(* Schneider Machine Expert - Basic project Ladder_Code, file version 2.7.0.0 *)
(* ProjectInformations: Name=New project *)

HARDWARE
  Cpu 0: TM200CE40R
  EthernetConfiguration: NetworkName=M200, IpAllocationMode=FixedAddress, IpAddress=192.168.1.200, SubnetMask=255.255.255.0
  SerialLineConfiguration: Baud=Baud19200, Parity=ParityEven, DataBits=DataBits8, StopBits=StopBits1, PhysicalMedium=PhysicalMediumRs485, TransmissionMode=TransmissionModeModbusRtu, SlaveId=1, Addressing=MasterAddressing
  MastTask: UsePeriodScanMode=false, PeriodScan=100
  FastTask: Period=255
  CpuBehavior: StartingMode=StartAsPreviousState, AutoSaveRamOnEeprom=true, WatchdogPeriod=250

SYMBOLS  (address, symbol, comment, settings)
  %TM0        [Type=TP, Preset=1, Base=OneHundredMilliSeconds]
  %TM1        [Type=TP, Preset=1, Base=OneHundredMilliSeconds]
  %READ_VAR0   [Link(Value(FBComLinkParameterEnums=SerialLine1)), RemoteDeviceId(Value(int=1)), Timeout(Value(int=100)), ObjType(Value(FBComObjTypeParameterEnums=MW)), FirstObj(Value(int=0)), Quantity(Value(int=1)), IndexData(Value(int=100))]
  %WRITE_VAR0   [Link(Value(FBComLinkParameterEnums=SerialLine1)), RemoteDeviceId(Value(int=1)), Timeout(Value(int=100)), ObjType(Value(FBComObjTypeParameterEnums=MW)), FirstObj(Value(int=1)), Quantity(Value(int=1)), IndexData(Value(int=1))]

POU New POU
  (* SectionNumber=1 *)

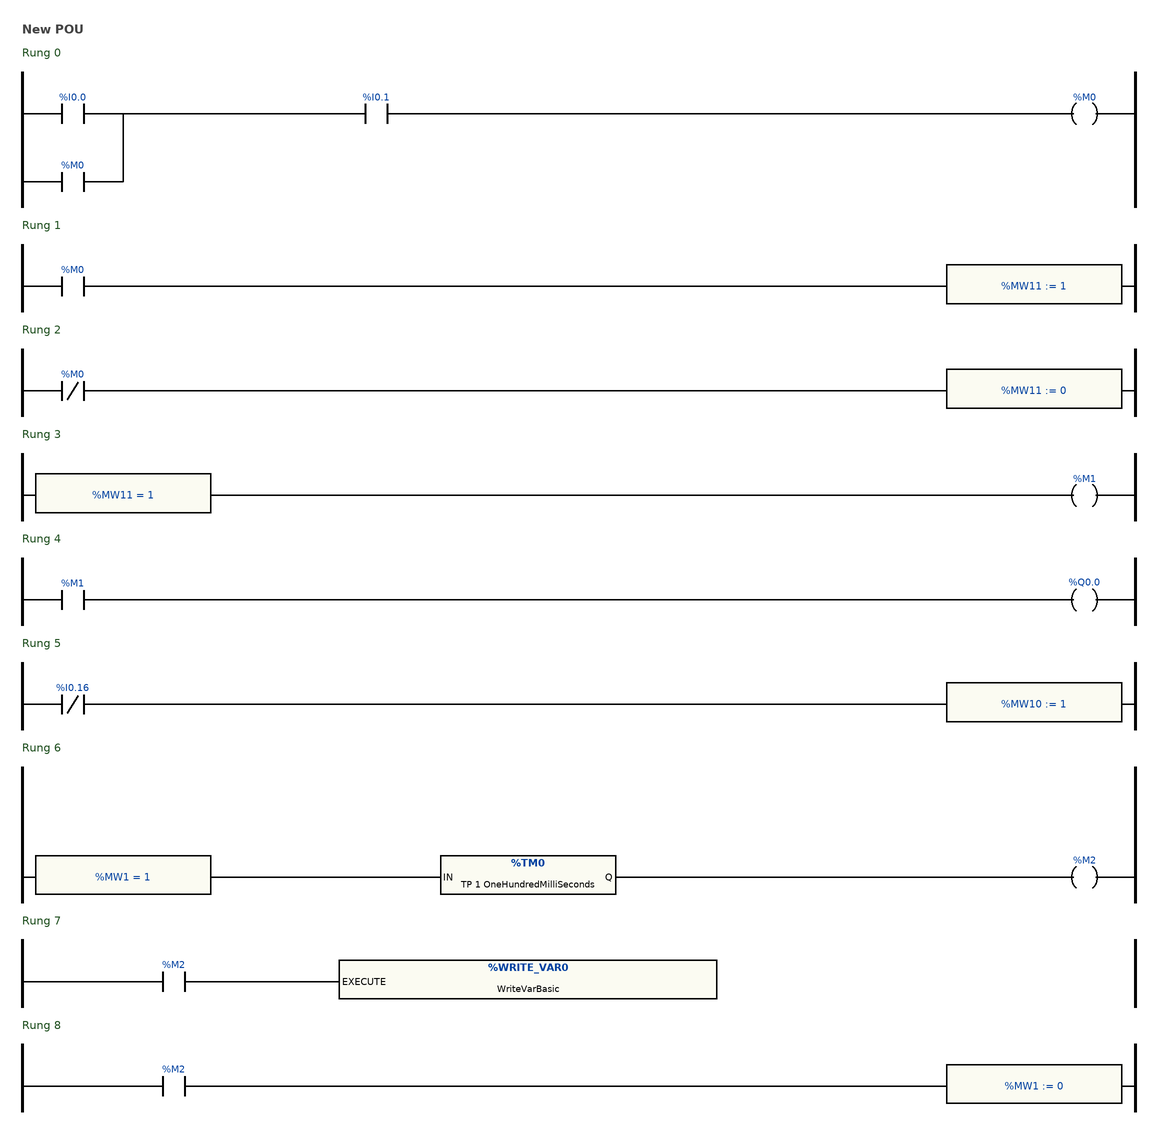

// Rung 0
  LD %I0.0
  OR %M0
  AND %I0.1
  ST %M0
  // as ST:
  //   %M0 := (%I0.0 OR %M0) AND %I0.1;

// Rung 1
  LD %M0
  [ %MW11 := 1 ]
  // as ST:
  //   IF %M0 THEN %MW11 := 1; END_IF;

// Rung 2
  LDN %M0
  [ %MW11 := 0 ]
  // as ST:
  //   IF NOT %M0 THEN %MW11 := 0; END_IF;

// Rung 3
  LD [ %MW11 = 1 ]
  ST %M1
  // as ST:
  //   %M1 := %MW11 = 1;

// Rung 4
  LD %M1
  ST %Q0.0
  // as ST:
  //   %Q0.0 := %M1;

// Rung 5
  LDN %I0.16
  [ %MW10 := 1 ]
  // as ST:
  //   IF NOT %I0.16 THEN %MW10 := 1; END_IF;

// Rung 6
  BLK %TM0
  LD [ %MW1 = 1 ]
  IN
  OUT_BLK
  LD Q
  ST %M2
  END_BLK
  // as ST:
  //   %TM0(IN := %MW1 = 1);
  //   %M2 := %TM0.Q;

// Rung 7
  BLK %WRITE_VAR0
  LD %M2
  EXECUTE
  END_BLK
  // as ST:
  //   %WRITE_VAR0(EXECUTE := %M2);

// Rung 8
  LD %M2
  [ %MW1 := 0 ]
  // as ST:
  //   IF %M2 THEN %MW1 := 0; END_IF;

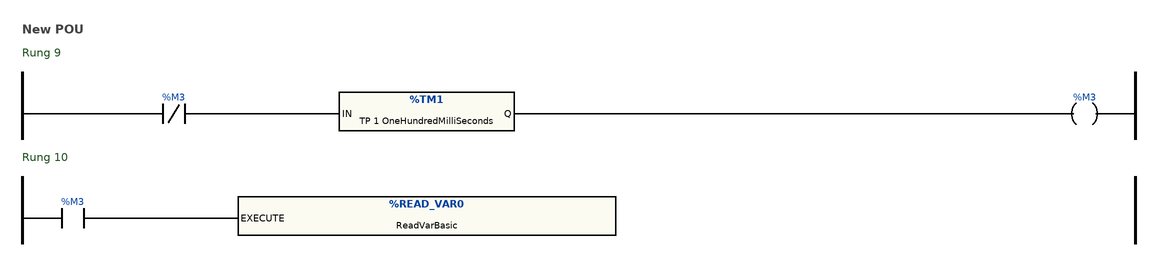

// Rung 9
  BLK %TM1
  LDN %M3
  IN
  OUT_BLK
  LD Q
  ST %M3
  END_BLK
  // as ST:
  //   %TM1(IN := NOT %M3);
  //   %M3 := %TM1.Q;

// Rung 10
  BLK %READ_VAR0
  LD %M3
  EXECUTE
  END_BLK
  // as ST:
  //   %READ_VAR0(EXECUTE := %M3);
